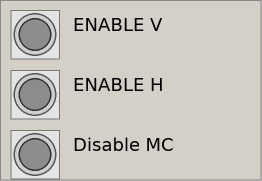
VISUALIZATION IO  // 262x181
    PushSwitchLed (10,10 50x49), variable: MAIN.limitEnable1, behaviour: TOGGLE, style: Switch-PushSwitchLed-Gray
    PushSwitchLed (10,70 50x49), variable: MAIN.limitEnable2, behaviour: TOGGLE, style: Switch-PushSwitchLed-Gray
    Label (70,10 190x30), "ENABLE V"
    Label (70,70 190x30), "ENABLE H"
    PushSwitchLed (10,130 50x49), variable: MAIN.bDisableMC, behaviour: TOGGLE, style: Switch-PushSwitchLed-Gray
    Label (70,130 190x30), "Disable MC"
END_VISUALIZATION

(* stored: Version 1.1.0.1, ProductVersion 3.1.4022.12
   Visu IO: Id {9dc0ac37-2bf6-4796-b628-6664538793f0} *)
